Fanuc KAREL source: ko00106.KL

-- PROVISIONAL review KL for V1013-1; original PC SHA256 3eeef7421de833f49a35bd30f75c3dc54baa663998b2cf794c4ef25d02bb0c40
-- Incomplete behavior may be omitted. Consult companion uncertainty JSON. Do not deploy.
PROGRAM KO00106
%NOLOCKGROUP
VAR
  A : REAL
  B : INTEGER
  OUT : REAL
BEGIN
  -- UNRESOLVED_PC offsets 5-13; opcodes 9D,64,23
  -- UNRESOLVED_PC offsets 18-29; opcodes 2E,23
  -- UNRESOLVED_PC offsets 34-57; opcodes 27,22,27,21,64,76,23
  -- UNRESOLVED_PC offsets 62-66; opcodes 7F
END KO00106
